// TwinCAT 3 PLC project PlcAxis
// ProgramVersion: 3.1.4024.0
// libraries:
//   Tc2_Math, * (Beckhoff Automation GmbH)
// project tree:
//   POUs/ MAIN.TcPOU

// ---- POUs/MAIN.TcPOU
PROGRAM MAIN
VAR
    rawPosition : LREAL;
    wrappedAngle : LREAL;
    signedAngle : LREAL;
    wholeTurns : LREAL;
    turnFraction : LREAL;
END_VAR

rawPosition := rawPosition + 400.56;
wrappedAngle := MODABS(rawPosition, 360.0);
signedAngle := LMOD(rawPosition, 360.0);
wholeTurns := LTRUNC(rawPosition / 360.0);
turnFraction := FRAC(rawPosition / 360.0);

END_PROGRAM
